SUBAPPLICATION ACTION_SERVER_FEEDBACK_MESSAGE
  (* Standard: 61499-2 *)
  (* Version 1.0, 2023-04-02, Tim Hesse *)
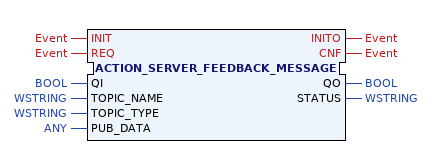
  EVENT_INPUT
    INIT; (* Initialization Request *)
    REQ;
  END_EVENT
  EVENT_OUTPUT
    INITO; (* Initialization Confirm *)
    CNF;
  END_EVENT
  VAR_INPUT
    QI : BOOL; (* Input event qualifier *)
    TOPIC_NAME : WSTRING;
    TOPIC_TYPE : WSTRING;
    PUB_DATA : ANY;
  END_VAR
  VAR_OUTPUT
    QO : BOOL; (* Output event qualifier *)
    STATUS : WSTRING;
  END_VAR
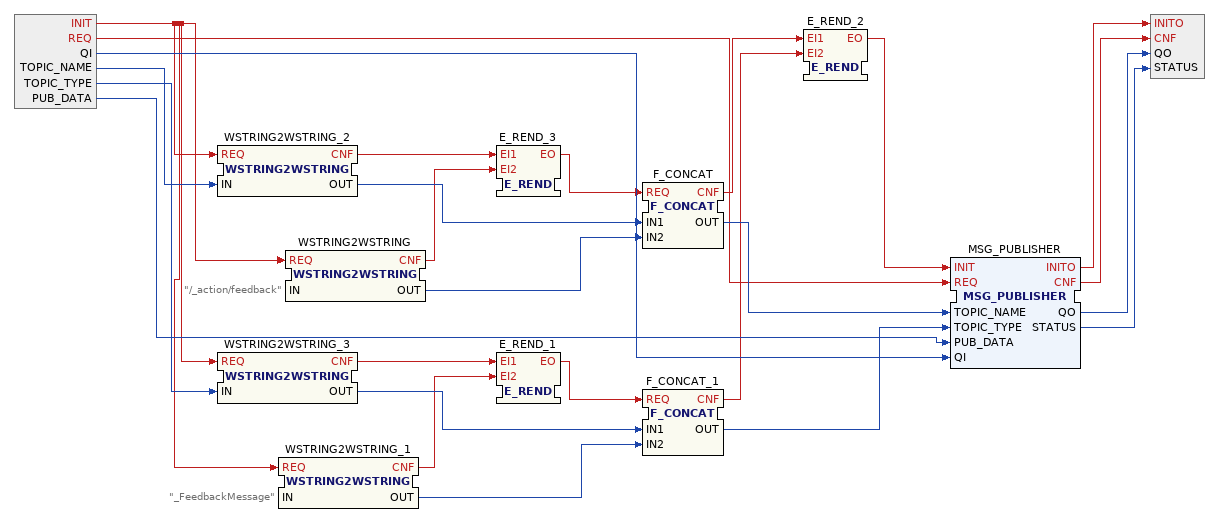
  FBS
    WSTRING2WSTRING : WSTRING2WSTRING(IN := "/_action/feedback");
    E_REND_3 : E_REND;
    WSTRING2WSTRING_1 : WSTRING2WSTRING(IN := "_FeedbackMessage");
    F_CONCAT : F_CONCAT;
    WSTRING2WSTRING_3 : WSTRING2WSTRING;
    E_REND_2 : E_REND;
    WSTRING2WSTRING_2 : WSTRING2WSTRING;
    E_REND_1 : E_REND;
    F_CONCAT_1 : F_CONCAT;
  END_FBS
  SUBAPPS
    MSG_PUBLISHER : MSG_PUBLISHER;
  END_SUBAPPS
  EVENT_CONNECTIONS
    WSTRING2WSTRING_3.CNF TO E_REND_1.EI1;
    F_CONCAT.CNF TO E_REND_2.EI1;
    F_CONCAT_1.CNF TO E_REND_2.EI2;
    WSTRING2WSTRING_1.CNF TO E_REND_1.EI2;
    E_REND_1.EO TO F_CONCAT_1.REQ;
    WSTRING2WSTRING_2.CNF TO E_REND_3.EI1;
    E_REND_3.EO TO F_CONCAT.REQ;
    WSTRING2WSTRING.CNF TO E_REND_3.EI2;
    E_REND_2.EO TO MSG_PUBLISHER.INIT;
    INIT TO WSTRING2WSTRING_2.REQ;
    INIT TO WSTRING2WSTRING_3.REQ;
    INIT TO WSTRING2WSTRING_1.REQ;
    INIT TO WSTRING2WSTRING.REQ;
    REQ TO MSG_PUBLISHER.REQ;
    MSG_PUBLISHER.INITO TO INITO;
    MSG_PUBLISHER.CNF TO CNF;
  END_CONNECTIONS
  DATA_CONNECTIONS
    WSTRING2WSTRING_3.OUT TO F_CONCAT_1.IN1;
    WSTRING2WSTRING_2.OUT TO F_CONCAT.IN1;
    WSTRING2WSTRING_1.OUT TO F_CONCAT_1.IN2;
    WSTRING2WSTRING.OUT TO F_CONCAT.IN2;
    F_CONCAT.OUT TO MSG_PUBLISHER.TOPIC_NAME;
    F_CONCAT_1.OUT TO MSG_PUBLISHER.TOPIC_TYPE;
    TOPIC_NAME TO WSTRING2WSTRING_2.IN;
    TOPIC_TYPE TO WSTRING2WSTRING_3.IN;
    PUB_DATA TO MSG_PUBLISHER.PUB_DATA;
    QI TO MSG_PUBLISHER.QI;
    MSG_PUBLISHER.QO TO QO;
    MSG_PUBLISHER.STATUS TO STATUS;
  END_CONNECTIONS
END_SUBAPPLICATION
